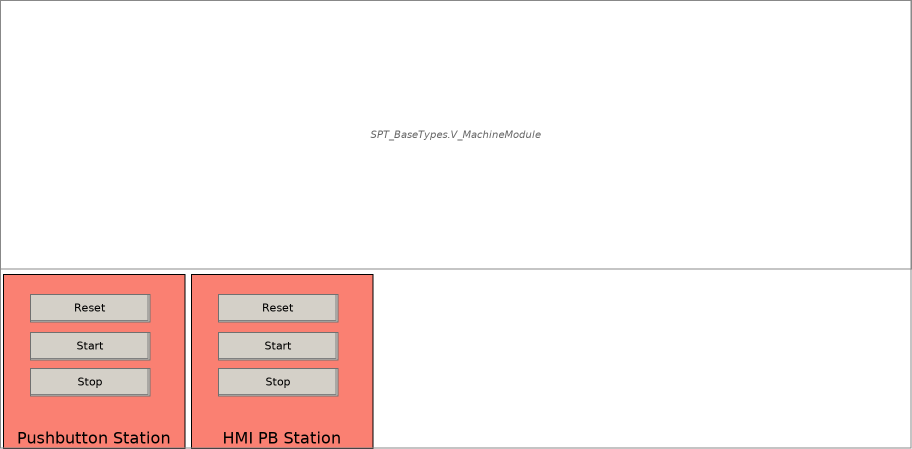
VISUALIZATION V_Main  // 912x449
    Frame (0,0 912x269)
        shows SPT_BaseTypes.V_MachineModule(HMI := MAIN.XPlanarModule.PackMLBaseModule_HMI)
    Group (3,274 182x175)
        RoundedRectangle (0,0 182x175), "Pushbutton Station"
        Button (27,94 120x28), "Stop", input disabled if: not MAIN.ControlSourcePB.MainPMLControl_Simplified.StopPermissive
            tap MAIN.ControlSourcePB.MainPMLControl_Simplified.StopPressed
        Button (27,20 120x28), "Reset", input disabled if: not MAIN.ControlSourcePB.MainPMLControl_Simplified.ResetPermissive
            tap MAIN.ControlSourcePB.MainPMLControl_Simplified.ResetPressed
        Button (27,58 120x28), "Start", input disabled if: not MAIN.ControlSourcePB.MainPMLControl_Simplified.StartPermissive
            tap MAIN.ControlSourcePB.MainPMLControl_Simplified.StartPressed
    Group (191,274 182x175)
        RoundedRectangle (0,0 182x175), "HMI PB Station"
        Button (27,94 120x28), "Stop", input disabled if: not MAIN.ControlSourceHMI.MainPMLControl_Simplified.StopPermissive
            tap MAIN.ControlSourceHMI.MainPMLControl_Simplified.StopPressed
        Button (27,20 120x28), "Reset", input disabled if: not MAIN.ControlSourceHMI.MainPMLControl_Simplified.ResetPermissive
            tap MAIN.ControlSourceHMI.MainPMLControl_Simplified.ResetPressed
        Button (27,58 120x28), "Start", input disabled if: not MAIN.ControlSourceHMI.MainPMLControl_Simplified.StartPermissive
            tap MAIN.ControlSourceHMI.MainPMLControl_Simplified.StartPressed
END_VISUALIZATION

(* stored: Version 1.1.0.1, ProductVersion 3.1.4024.13
   Visu V_Main: Id {a820fc1e-d71f-479f-a200-f2cc0d18dc0b} *)
